FUNCTION_BLOCK F_INT_TO_SINT (* Convert INT to SINT *)
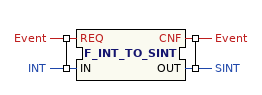
  EVENT_INPUT
    REQ WITH IN; (* Normal Execution Request *)
  END_EVENT
  EVENT_OUTPUT
    CNF WITH OUT; (* Execution Confirmation *)
  END_EVENT
  VAR_INPUT
    IN : INT;
  END_VAR
  VAR_OUTPUT
    OUT : SINT;
  END_VAR
END_FUNCTION_BLOCK
